{attribute 'qualified_only'}
TYPE E_MMVehicleCommand :
(
	eMMVehicleCommand_NoCommandInProgress 	:= 0,																	(**)
	eMMVehicleCommand_MoveVehicleToStation	:= 176,																	(**)
	eMMVehicleCommand_MoveVehicleToPosition	:= 177																	(**)
) BYTE;
END_TYPE

(* stored: Version 1.1.0.1, ProductVersion 3.1.4024.5
   EnumerationTextList E_MMVehicleCommand: Id {5b721bc1-05ee-4cb0-88b2-7ba009969c5d} *)
